// Mitsubishi GX Works2 project: ex2 group12_mostUpdate (4)   PLC: FX3G

// global labels: Global1
VAR_GLOBAL
  start_work_day AT X007 : BOOL;
  work_day_light AT Y000 : BOOL;
  end_the_day AT M7 : BOOL;
  alarm_switch AT X005 : BOOL;
  out_of_stock AT M3 : BOOL;
  honey_container AT D1121 : REAL;
  mixing AT D1131 : REAL;
  baking AT D1141 : REAL;
  oat_input AT D1161 : REAL;
  protein_input AT D1171 : REAL;
  honey_input AT D1181 : REAL;
  input_light AT M2 : BOOL;
  save_analog AT D1151 : REAL;
  sample_analog_1 AT X003 : BOOL;
END_VAR
VAR_GLOBAL CONSTANT
  const_400 : REAL := 400;
  const_320 : REAL := 320;
  const_160 : REAL := 160;
END_VAR
VAR_GLOBAL
  normalized_input AT D1191 : REAL;
END_VAR
VAR_GLOBAL CONSTANT
  const_6 : REAL := 6;
  const_5 : REAL := 5;
END_VAR
VAR_GLOBAL
  choose_protein AT M6 : BOOL;
  choose_classic AT M5 : BOOL;
END_VAR
VAR_GLOBAL CONSTANT
  const_float_400 : REAL := 400;
  const_word_320 : REAL := 320;
  const_word_160 : REAL := 160;
END_VAR
VAR_GLOBAL
  oats_container AT D1101 : REAL;
  proteins_container AT D1111 : REAL;
END_VAR
VAR_GLOBAL CONSTANT
  const_word_240 : REAL := 240;
END_VAR
VAR_GLOBAL
  finish_moving AT M4 : BOOL;
END_VAR
VAR_GLOBAL CONSTANT
  const_word_120 : INT := 120;
END_VAR
VAR_GLOBAL
  TC_1 AT TC1 : BOOL;
END_VAR
VAR_GLOBAL CONSTANT
  const_50_mix : INT := 50;
END_VAR
VAR_GLOBAL
  mixing_light AT Y003 : BOOL;
  TS_1 AT TS1 : BOOL;
  switch_mix_to_bake AT X002 : BOOL;
  cbaking_timer_c AT TS2 : BOOL;
  TC_2 AT TC2 : BOOL;
END_VAR
VAR_GLOBAL CONSTANT
  const_40_bake_c : INT := 40;
END_VAR
VAR_GLOBAL
  TC_3 AT TC3 : BOOL;
END_VAR
VAR_GLOBAL CONSTANT
  const_50_bake_p : INT := 50;
END_VAR
VAR_GLOBAL
  baking_light AT M8 : BOOL;
  baking_timer_c AT TS2 : BOOL;
  baking_timer_p AT TS3 : BOOL;
  TRY AT D1176 : REAL;
  flickering_light AT M9 : BOOL;
  TC_4 AT TC4 : BOOL;
END_VAR
VAR_GLOBAL CONSTANT
  const_5_light : INT := 5;
END_VAR
VAR_GLOBAL
  Y1_timer AT TS4 : BOOL;
  baking_light_1 AT Y001 : BOOL;
  baking_light_2 AT Y002 : BOOL;
  Y2_timer AT TS5 : BOOL;
END_VAR
VAR_GLOBAL CONSTANT
  const_f_680 : INT := 680;
END_VAR
VAR_GLOBAL
  save_mixing AT D1191 : REAL;
END_VAR
VAR_GLOBAL CONSTANT
  const_680 : REAL := 680;
END_VAR
VAR_GLOBAL
  TRY1 AT D1179 : REAL;
  start_packing AT X006 : BOOL;
  count_snack AT X000 : BOOL;
  pack_single_snack AT CC0 : BOOL;
END_VAR
VAR_GLOBAL CONSTANT
  const_single_snack : INT := 1;
END_VAR
VAR_GLOBAL
  packing_light AT Y004 : BOOL;
  pack_package AT CC1 : BOOL;
END_VAR
VAR_GLOBAL CONSTANT
  cont_package : INT := 8;
END_VAR
VAR_GLOBAL
  package_container AT D1200 : REAL;
END_VAR
VAR_GLOBAL CONSTANT
  const_single_package : REAL := 1;
END_VAR
VAR_GLOBAL
  pack_package_cs AT CS1 : BOOL;
  pack_single_cs AT CS0 : BOOL;
  storage AT D1210 : REAL;
END_VAR
VAR_GLOBAL CONSTANT
  const_40 : REAL := 40;
END_VAR
VAR_GLOBAL
  print_answer AT D1220 : REAL;
END_VAR
VAR_GLOBAL CONSTANT
  consconst_word_160t_word_160 : REAL := 400;
  const_240 : REAL := 240;
  const_120 : REAL := 120;
END_VAR
VAR_GLOBAL
  TC_five AT TC5 : BOOL;
  analog_output AT D8282 : INT;
  analog_input1 AT D8280 : INT;
  Try123 AT X011 : BOOL;
  iteration AT M2 : BOOL;
  mixing_light_time AT M13 : BOOL;
  new_stock AT M14 : BOOL;
END_VAR
VAR_GLOBAL CONSTANT
  const_0 : REAL;
  const_9 : INT := 9;
END_VAR

// task Task_01 (event TRUE, interval 0, priority 31): POU_01

PROGRAM POU_01
VAR
  analog_input_1 : INT;
  save_analog_input : REAL;
  save_analog_1 : REAL;
  TC_5 : BOOL;
END_VAR
(* structured ladder/FBD written out as ST: instructions are called as NAME(EN, inputs, outputs); _pN, _eN, _tN stand for wires *)
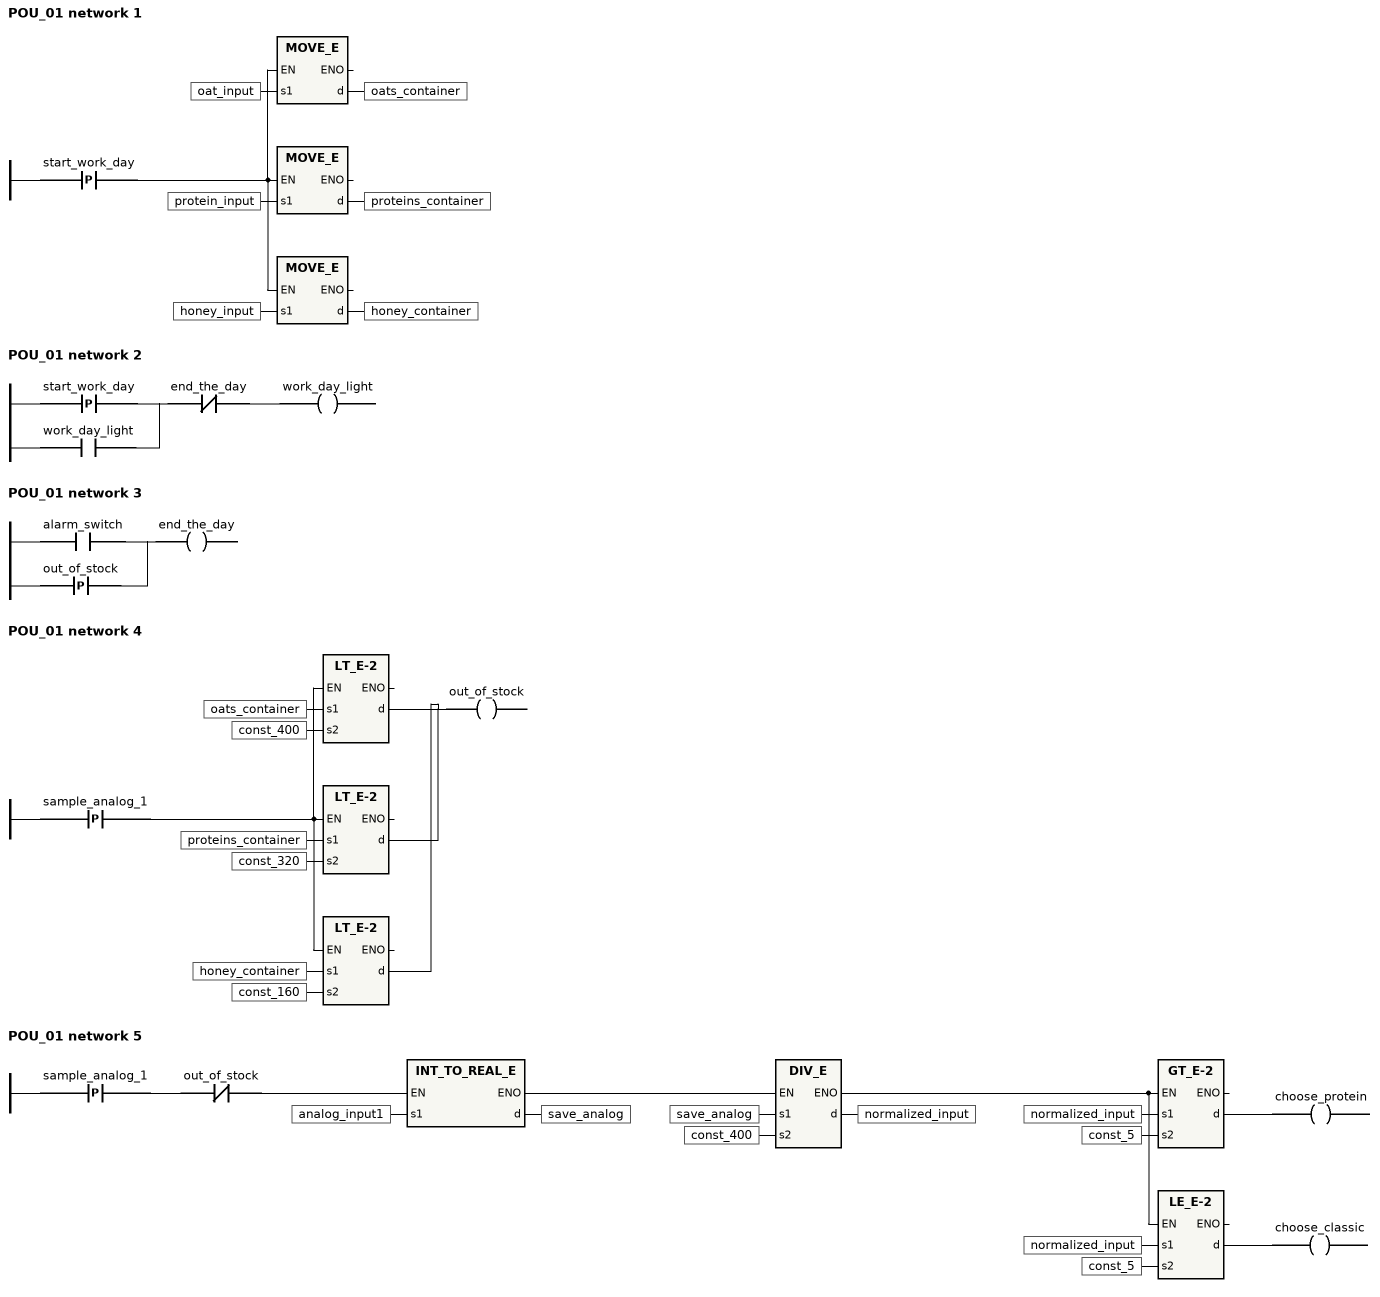
(* network 1 *)
_p1 := LDP(TRUE, start_work_day);
MOVE_E(_p1, oat_input, oats_container);
MOVE_E(_p1, protein_input, proteins_container);
MOVE_E(_p1, honey_input, honey_container);
(* network 2 *)
work_day_light := (LDP(TRUE, start_work_day) OR work_day_light) AND NOT end_the_day;
(* network 3 *)
end_the_day := alarm_switch OR LDP(TRUE, out_of_stock);
(* network 4 *)
_p1 := LDP(TRUE, sample_analog_1);
LT_E(_p1, oats_container, const_400, _t2);
LT_E(_p1, proteins_container, const_320, _t3);
LT_E(_p1, honey_container, const_160, _t4);
out_of_stock := _t2 OR _t3 OR _t4;
(* network 5 *)
_e1 := INT_TO_REAL_E(LDP(TRUE, sample_analog_1) AND NOT out_of_stock, analog_input1, save_analog);
_e2 := DIV_E(_e1, save_analog, const_400, normalized_input);
GT_E(_e2, normalized_input, const_5, _t3);
choose_protein := _t3;
LE_E(_e2, normalized_input, const_5, _t4);
choose_classic := _t4;
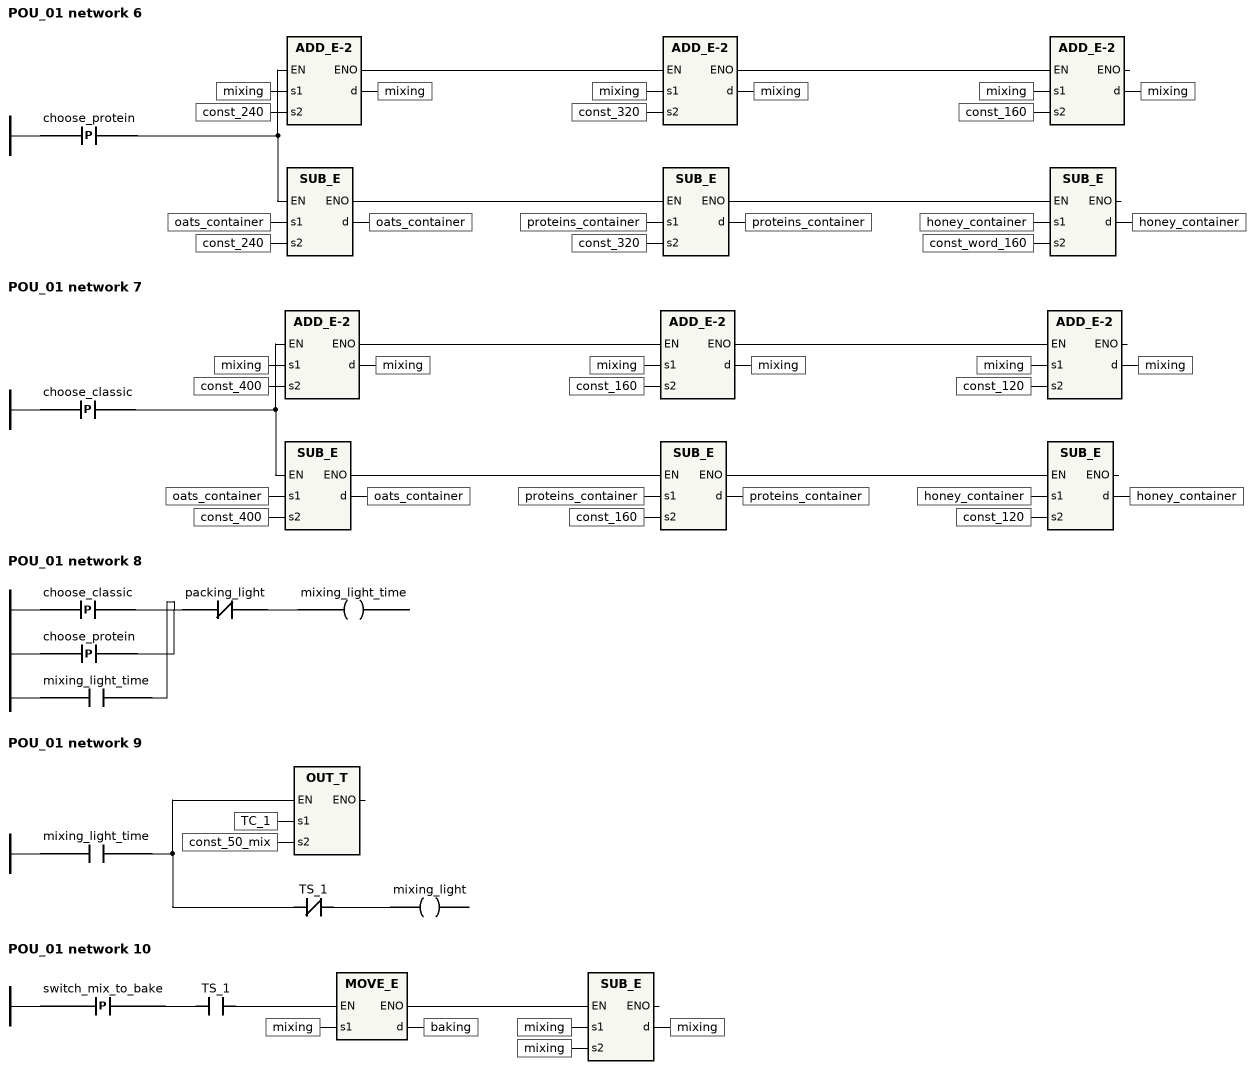
(* network 6 *)
_p1 := LDP(TRUE, choose_protein);
_e2 := ADD_E(_p1, mixing, const_240, mixing);
_e3 := ADD_E(_e2, mixing, const_320, mixing);
ADD_E(_e3, mixing, const_160, mixing);
_e4 := SUB_E(_p1, oats_container, const_240, oats_container);
_e5 := SUB_E(_e4, proteins_container, const_320, proteins_container);
SUB_E(_e5, honey_container, const_word_160, honey_container);
(* network 7 *)
_p1 := LDP(TRUE, choose_classic);
_e2 := ADD_E(_p1, mixing, const_400, mixing);
_e3 := ADD_E(_e2, mixing, const_160, mixing);
ADD_E(_e3, mixing, const_120, mixing);
_e4 := SUB_E(_p1, oats_container, const_400, oats_container);
_e5 := SUB_E(_e4, proteins_container, const_160, proteins_container);
SUB_E(_e5, honey_container, const_120, honey_container);
(* network 8 *)
mixing_light_time := (LDP(TRUE, choose_classic) OR LDP(TRUE, choose_protein) OR mixing_light_time) AND NOT packing_light;
(* network 9 *)
OUT_T(mixing_light_time, TC_1, const_50_mix);
mixing_light := mixing_light_time AND NOT TS_1;
(* network 10 *)
_e1 := MOVE_E(LDP(TRUE, switch_mix_to_bake) AND TS_1, mixing, baking);
SUB_E(_e1, mixing, mixing, mixing);
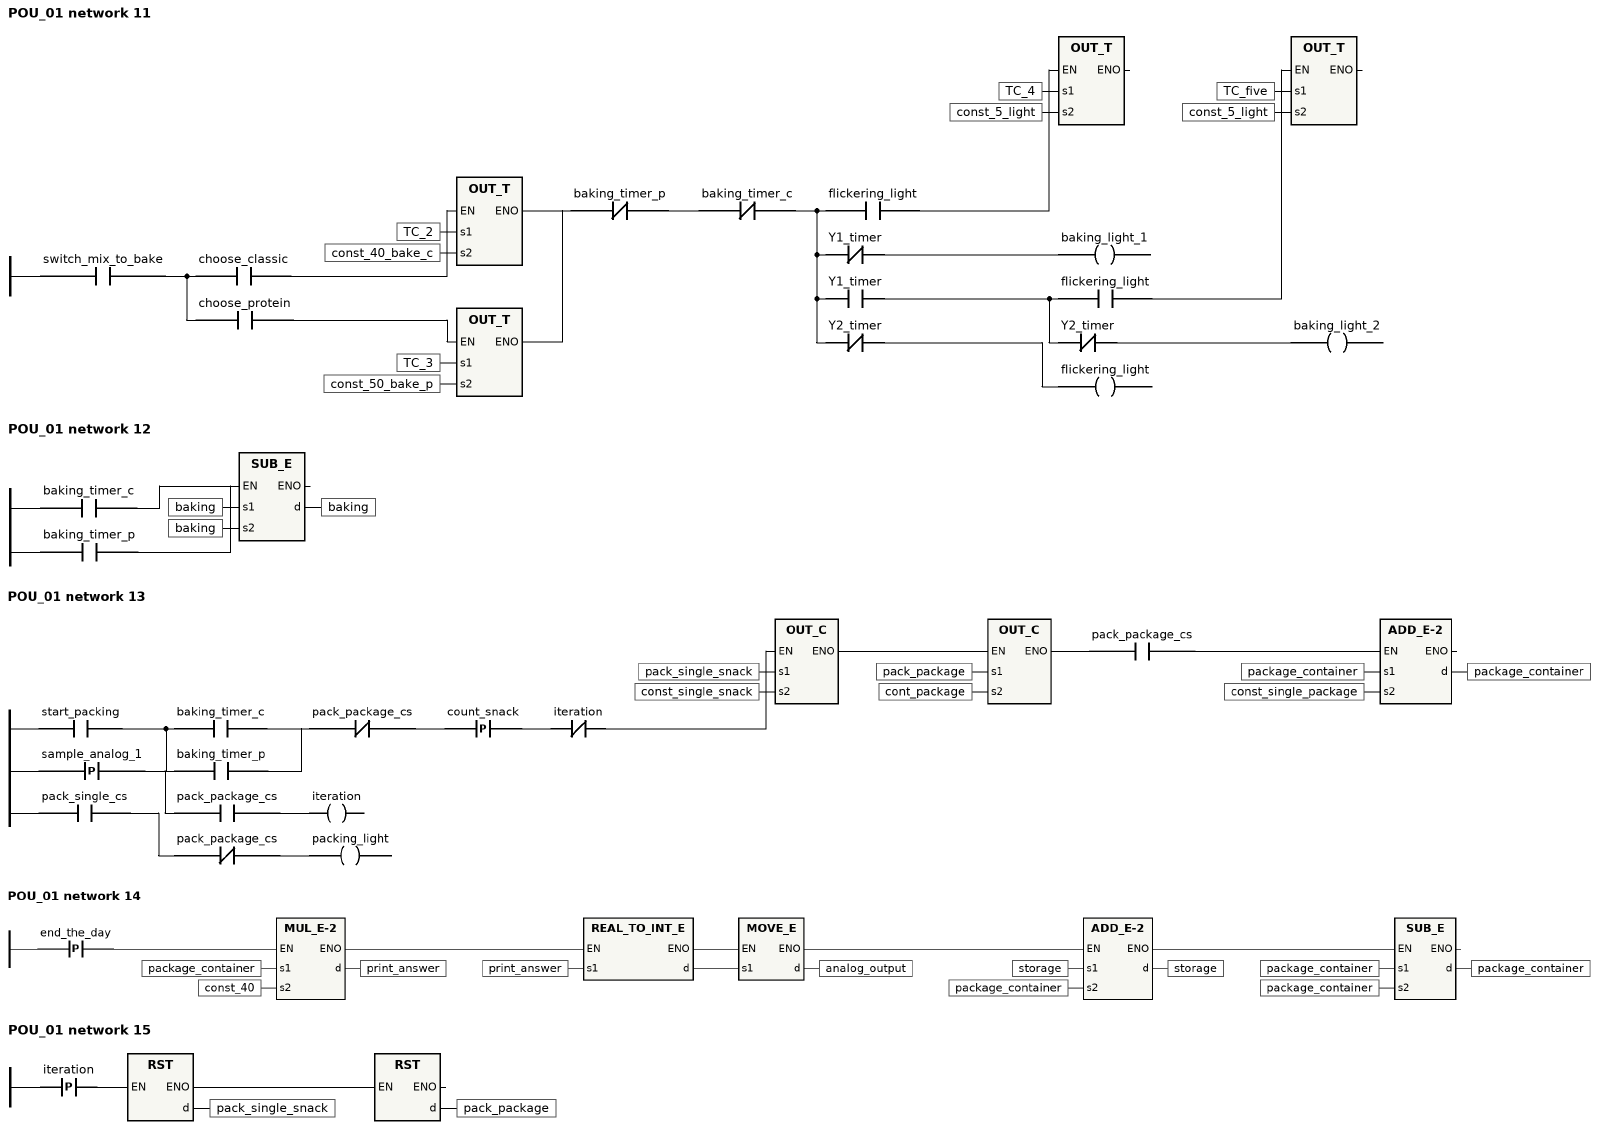
(* network 11 *)
_e1 := OUT_T(switch_mix_to_bake AND choose_classic, TC_2, const_40_bake_c);
_e2 := OUT_T(switch_mix_to_bake AND choose_protein, TC_3, const_50_bake_p);
_p3 := ((_e1 OR _e2) AND NOT baking_timer_p) AND NOT baking_timer_c;
OUT_T(_p3 AND flickering_light, TC_4, const_5_light);
baking_light_1 := _p3 AND NOT Y1_timer;
_p4 := _p3 AND Y1_timer;
OUT_T(_p4 AND flickering_light, TC_five, const_5_light);
baking_light_2 := _p4 AND NOT Y2_timer;
flickering_light := _p3 AND NOT Y2_timer;
(* network 12 *)
SUB_E(baking_timer_c OR baking_timer_p, baking, baking, baking);
(* network 13 *)
_e1 := OUT_C(((((start_packing AND baking_timer_c) OR (start_packing AND baking_timer_p)) AND NOT pack_package_cs) AND LDP(TRUE, count_snack)) AND NOT iteration, pack_single_snack, const_single_snack);
_e2 := OUT_C(_e1, pack_package, cont_package);
ADD_E(_e2 AND pack_package_cs, package_container, const_single_package, package_container);
iteration := LDP(TRUE, sample_analog_1) AND pack_package_cs;
packing_light := pack_single_cs AND NOT pack_package_cs;
(* network 14 *)
_e1 := MUL_E(LDP(TRUE, end_the_day), package_container, const_40, print_answer);
_e3 := REAL_TO_INT_E(_e1, print_answer, _t2);
_e4 := MOVE_E(_e3, _t2, analog_output);
_e5 := ADD_E(_e4, storage, package_container, storage);
SUB_E(_e5, package_container, package_container, package_container);
(* network 15 *)
_e1 := RST(LDP(TRUE, iteration), pack_single_snack);
RST(_e1, pack_package);
END_PROGRAM
